SYSTEM Empty
  (* Version 1.0, 2007-10-25, Goran Cengic, Chalmers *)
  DEVICE Test Device : DeviceType_not_used
    RESOURCE Test Resource : ResourceType_not_used
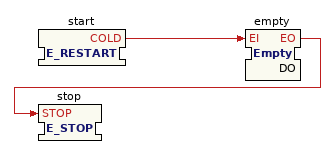
      FBS
        start : E_RESTART;
        stop : E_STOP;
        empty : Empty;
      END_FBS
      EVENT_CONNECTIONS
        start.COLD TO empty.EI;
        empty.EO TO stop.STOP;
      END_CONNECTIONS
    END_RESOURCE
  END_DEVICE
END_SYSTEM
